// TIA Portal V21 export
FUNCTION "GestioneMacchina_010102" : Void   // FC147, LAD
{ S7_Optimized_Access := 'TRUE' }
// stored: SetENOAutomatically false
BEGIN
END_FUNCTION
